FUNCTION_BLOCK E_RESTART
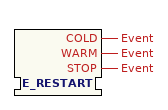
  EVENT_OUTPUT
    COLD;
    WARM;
    STOP;
  END_EVENT
END_FUNCTION_BLOCK
